{attribute addProperty BoxType "KL1908"}
{attribute addProperty Id "Channel_1Channel_D8611DE600"}
{attribute addProperty CRC "1578653816"}
{attribute addProperty SizeInBites "0"}
{attribute addProperty SizeInBytes "0"}
TYPE KL1908_5E185878 :
STRUCT
	{attribute addProperty Name "Channel_1"}
	Channel_1 : Channel_D8611DE6;
END_STRUCT
END_TYPE

(* stored: Version 1.2.0.0, ProductVersion 3.1.4024.9
   DUT KL1908_5E185878: Id {d1fe7ee5-17d0-4f51-8289-2e355a033485} *)
